{attribute 'qualified_only'}
{attribute 'strict'}
TYPE E_CabinetJob :
(
	Idle :=0,
	Initial,
	MoveIn,
	MoveOut,
	MovingOut,
	MovingIn,
	Moved,
	Finish,
	Error
);
END_TYPE

(* stored: Version 1.1.0.1, ProductVersion 3.1.4024.13
   DUT E_CabinetJob: Id {f3c83675-19a4-4d87-adae-653505ebbe09} *)
